INTERFACE IEventHandler_OnMinutesChanged EXTENDS IEventHandlerBase

METHOD OnMinutesChanged
VAR_INPUT
	Now: TIMESTRUCT;
END_VAR
END_METHOD

END_INTERFACE

(* stored: Version 1.1.0.1, ProductVersion 3.1.4024.3
   Itf IEventHandler_OnMinutesChanged: Id {3673e252-4e05-0b95-34ca-b1a4cfa0cb35}
   Method OnMinutesChanged: Id {65c67529-cc6c-06cf-0141-05a27cf82737} *)
